FUNCTION_BLOCK CraneAngle
VAR_INPUT
	par : ST_pValveControlledCylinder;
	a : LREAL;
	b : LREAL;
	c : LREAL;
END_VAR
VAR_OUTPUT
	thetaAngle : LREAL;
END_VAR
VAR
    thetaAngleRad : LREAL;
	thetaAngleDeg : LREAL;
END_VAR


//Angle A joint 1 and joint 2
thetaAngle := ACOS( (EXPT(b,2) + EXPT(c,2) - EXPT(a,2) ) / ((2) * b * c));

//To make it into degrees if i need that:
thetaAngleDeg := thetaAngle*(180/par.pi);

END_FUNCTION_BLOCK

(* stored: Version 1.1.0.1, ProductVersion 3.1.4024.9
   POU CraneAngle: Id {9659ca86-e779-4b60-b3a4-04e044f00676}, SpecialFunc None *)
